// TIA Portal V19 export
DATA_BLOCK "EmNodes"   // DB57
// stored: Access Published, MemoryReserve 100, Namespace Unit3
   VAR
      unitStatus { ExternalWritable := 'False'} : "LAF_typeUnitStatus";   // Status of the unit
      emFeedback { ExternalWritable := 'False'} : Array[0.._.Unit3_NO_OF_EMs] of "LUC_typeEmFeedback";   // Status of the individual equipment modules
      emRelations { ExternalWritable := 'False'} : Struct   // This is an example
         EM1 : Struct
            readyToReceive : Bool;
            readyToDeliver : Bool;
         END_STRUCT;
         EM2 : Struct
            readyToReceive : Bool;
            readyToDeliver : Bool;
         END_STRUCT;
         EM3 : Struct
            readyToReceive : Bool;
            readyToDeliver : Bool;
         END_STRUCT;
         EM4 : Struct
            readyToReceive : Bool;
            readyToDeliver : Bool;
         END_STRUCT;
      END_STRUCT;
      signalStack { ExternalWritable := 'False'} : "LUC_typeSignalStackByBool";
      emStatus : Array[0.._.Unit3_NO_OF_EMs] of "LUC_typeStates";
   END_VAR
BEGIN
END_DATA_BLOCK
